Universal Robots PolyScope program: Place_program.urp

Program Place_program (installation=default directory=/ursim/programs/MQTT createdIn=5.16.0 lastSavedIn=5.16.0 robotSerialNumber=20195599999)
Calibrated DH parameters: a=[0, -0.425, -0.3922, 0, 0, 0]; d=[0.1625, 0, 0, 0.1333, 0.0997, 0.0996]; alpha=[1.570796, 0, 0, 1.570796, -1.570796, 0]; deltaTheta=[0, 0, 0, 0, 0, 0]
InitVariablesNode variables(variable(name=cmd_name, expression=""), variable(name=object, expression=" "), variable(name=params, expression=" "), variable(name=topic_order, expression="robot/order"))
BeforeStart
  MoveJ speed 60 deg/s, acceleration 80 deg/s^2 (useActiveTCP=true) feature=Base
    Waypoint waiting_point_1: TCP in base x=492.803 y=288.649 z=418.324 mm, rx=2.6568 ry=-1.6608 rz=-0.0199 rad; joints [192.415, -98.238, 124.325, -115.253, -89.954, -13.481] deg
  object := "Pen"
Robot Program (runOnlyOnce=true)
  If object ≠ " "
    MoveJ speed 60 deg/s, acceleration 80 deg/s^2 (useActiveTCP=true) feature=Base
      Waypoint point_place: TCP in base x=807.912 y=-433.125 z=201.587 mm, rx=-0.6852 ry=3.024 rz=-0.0161 rad; joints [140.573, -55.8, 96.757, -132.886, -88.708, 25.083] deg
    MoveJ speed 60 deg/s, acceleration 80 deg/s^2 (useActiveTCP=true) feature=Base
      Waypoint waiting_point_2: TCP in base x=492.803 y=288.649 z=418.324 mm, rx=2.6568 ry=-1.6608 rz=-0.0199 rad; joints [192.415, -98.238, 124.325, -115.253, -89.954, -13.481] deg
  object := " "
